FUNCTION_BLOCK Section5
  (* Standard: 61499-2 *)
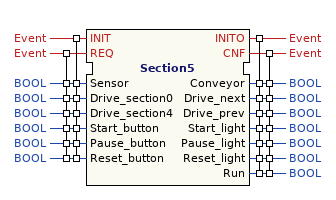
  EVENT_INPUT
    INIT WITH Sensor, Drive_section0, Drive_section4, Start_button, Pause_button, Reset_button;
    REQ WITH Sensor, Drive_section0, Drive_section4, Start_button, Pause_button, Reset_button;
  END_EVENT
  EVENT_OUTPUT
    INITO WITH Conveyor, Drive_next, Drive_prev, Start_light, Pause_light, Reset_light, Run;
    CNF WITH Conveyor, Drive_next, Drive_prev, Start_light, Pause_light, Reset_light, Run;
  END_EVENT
  VAR_INPUT
    Sensor : BOOL;
    Drive_section0 : BOOL;
    Drive_section4 : BOOL;
    Start_button : BOOL;
    Pause_button : BOOL;
    Reset_button : BOOL;
  END_VAR
  VAR_OUTPUT
    Conveyor : BOOL;
    Drive_next : BOOL;
    Drive_prev : BOOL;
    Start_light : BOOL;
    Pause_light : BOOL;
    Reset_light : BOOL;
    Run : BOOL;
  END_VAR
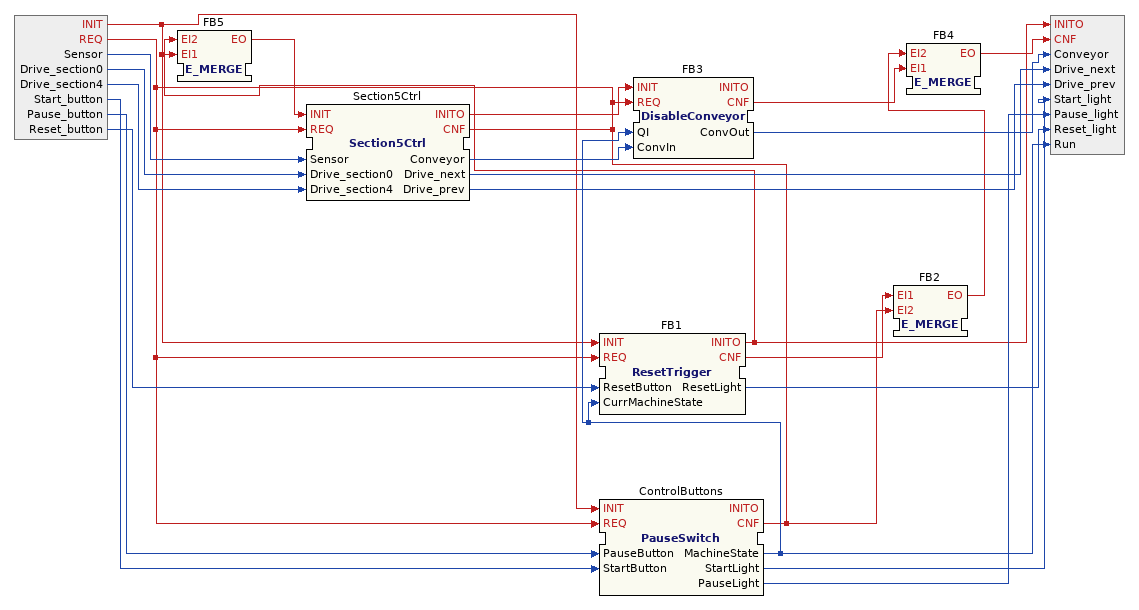
  FBS
    ControlButtons : PauseSwitch;
    FB1 : ResetTrigger;
    FB2 : E_MERGE;
    FB3 : DisableConveyor;
    FB4 : E_MERGE;
    Section5Ctrl : Section5Ctrl;
    FB5 : E_MERGE;
  END_FBS
  EVENT_CONNECTIONS
    INIT TO FB1.INIT;
    INIT TO ControlButtons.INIT;
    REQ TO FB1.REQ;
    REQ TO ControlButtons.REQ;
    FB1.INITO TO INITO;
    FB1.CNF TO FB2.EI1;
    ControlButtons.CNF TO FB2.EI2;
    REQ TO Section5Ctrl.REQ;
    Section5Ctrl.INITO TO FB3.INIT;
    REQ TO FB3.REQ;
    Section5Ctrl.CNF TO FB3.REQ;
    FB2.EO TO FB4.EI2;
    FB3.CNF TO FB4.EI1;
    FB4.EO TO CNF;
    ControlButtons.CNF TO FB3.REQ;
    FB1.INITO TO FB5.EI2;
    INIT TO FB5.EI1;
    FB5.EO TO Section5Ctrl.INIT;
  END_CONNECTIONS
  DATA_CONNECTIONS
    ControlButtons.MachineState TO FB1.CurrMachineState;
    Sensor TO Section5Ctrl.Sensor;
    Drive_section0 TO Section5Ctrl.Drive_section0;
    Drive_section4 TO Section5Ctrl.Drive_section4;
    Section5Ctrl.Conveyor TO FB3.ConvIn;
    Section5Ctrl.Drive_next TO Drive_next;
    Section5Ctrl.Drive_prev TO Drive_prev;
    FB3.ConvOut TO Conveyor;
    Start_button TO ControlButtons.StartButton;
    Pause_button TO ControlButtons.PauseButton;
    Reset_button TO FB1.ResetButton;
    ControlButtons.StartLight TO Start_light;
    ControlButtons.PauseLight TO Pause_light;
    FB1.ResetLight TO Reset_light;
    ControlButtons.MachineState TO Run;
    ControlButtons.MachineState TO FB3.QI;
  END_CONNECTIONS
END_FUNCTION_BLOCK
